FUNCTION_BLOCK ABSTRACT AttenuationFilterBase EXTENDS TExecution IMPLEMENTS IDevice
VAR_INPUT
END_VAR
VAR_OUTPUT
END_VAR
VAR
	{attribute 'OPC.UA.DA' := '0'}
	_name : STRING;
	{attribute 'OPC.UA.DA' := '0'}
	_deviceID : STRING;					
	{attribute 'OPC.UA.DA' := '0'}
	_family : DeviceFamily;				
	{attribute 'OPC.UA.DA' := '0'}
	_logger : Logger;
	{attribute 'OPC.UA.DA' := '0'}
	_message : StringBuilder;	
	{attribute 'OPC.UA.DA' := '0'}
	_attenuationFilterConfig : DeviceConfiguration;
END_VAR

PROPERTY DeviceID : STRING
GET
DeviceID := _deviceID;
END_GET
SET
_deviceID := DeviceID;
END_SET
END_PROPERTY

PROPERTY Family : DeviceFamily
GET
Family := _family;
END_GET
SET
_family := Family;
END_SET
END_PROPERTY

METHOD PROTECTED ABSTRACT GetPosition
VAR_INPUT
END_VAR
END_METHOD

METHOD PROTECTED ABSTRACT JogBackwardPosition
VAR_INPUT
	Execute : BOOL;
END_VAR
END_METHOD

METHOD PROTECTED ABSTRACT JogForwardPosition
VAR_INPUT
	Execute : BOOL;
END_VAR
END_METHOD

METHOD PROTECTED ABSTRACT MoveAbsPosition
VAR_INPUT
	Execute : BOOL;
	Position : LREAL;
END_VAR
END_METHOD

PROPERTY Name : STRING
GET
Name := _name;
END_GET
SET
_name := Name;
END_SET
END_PROPERTY

END_FUNCTION_BLOCK

(* stored: Version 1.1.0.1, ProductVersion 3.1.4024.4
   POU AttenuationFilterBase: Id {dd7a4ef9-a10f-405d-84c6-dad1f72da79f}, SpecialFunc None
   Property DeviceID: Id {5d50bbf3-fa60-4cf6-adc5-572a734da56d}
   Get Get: Id {13a4a7bc-326a-4732-a8d1-ae1515eacb26}
   Set Set: Id {850876c7-0dd4-4e2a-830f-be5bcc3ff908}
   Property Family: Id {448b9ded-eb01-4d87-83c4-d7c2db2547c2}
   Get Get: Id {859b4427-3c02-487a-a167-d054c3d58204}
   Set Set: Id {8fd65547-9a35-4dd7-8729-9af4da67a298}
   Method GetPosition: Id {f79182e7-0390-4987-b75c-f4afe43717de}
   Method JogBackwardPosition: Id {8a13cbaf-1e25-478c-88b1-36d38e43cf05}
   Method JogForwardPosition: Id {0c0c81ea-eb73-43b6-9fab-46ac17c18aca}
   Method MoveAbsPosition: Id {15f52c81-a33e-47b0-a424-a881848f174b}
   Property Name: Id {66243c01-1bb4-4101-8ba0-96d28b7809be}
   Get Get: Id {96815cef-e968-4499-811e-b5653834611e}
   Set Set: Id {b7e73377-bf8c-4b3d-b2e0-97e0cba7236c} *)
